INTERFACE ITF_MCRequiredChange EXTENDS ITF_IOButton

METHOD PUBLIC SetRequiredChange
VAR_INPUT
	bIn: BOOL;
END_VAR
END_METHOD

(*			
	RafalOS
	Rafał Osajda		04.11.2025		TC 4024.66
	
*)
METHOD Testing : BOOL
VAR_INPUT
END_VAR
END_METHOD

END_INTERFACE

(* stored: Version 1.1.0.1
   Itf ITF_MCRequiredChange: Id {0bb9e62f-bd86-08dc-230b-c32c9f5d16b2}
   Method SetRequiredChange: Id {5622f058-de00-0ab9-37a6-b85c4b833687}
   Method Testing: Id {727fa4b0-2551-05f9-3c28-0829bbfe35aa} *)
